// TIA Portal V16 program export: 1 tag tables, 0 data types, 3 data blocks, 1 code blocks (in call order from the OBs), 0 instance data blocks

VAR_GLOBAL   // PLC tag table "Default tag table"
   Web_Integer AT %MW10 : Int;
END_VAR

DATA_BLOCK "Data_block_1"   // DB1
{ S7_Optimized_Access := 'TRUE' }
VERSION : 0.1
// stored: AutoNumber true, DBAccessibleFromOPCUA true, IsOnlyStoredInLoadMemory false, IsRetainMemResEnabled false, IsWriteProtectedInAS false, MemoryReserve 100
   VAR
      in1 : Bool;
      in2 : Bool;
      in3 : Bool;
      out1 : Bool;
      out2 : Bool;
      out3 : Bool;
   END_VAR
BEGIN
END_DATA_BLOCK

DATA_BLOCK "Parameter_Control"   // DB2
{ S7_Optimized_Access := 'TRUE' }
// stored: MemoryReserve 100
   VAR
      Sugar : Real;
      Salt : Int;
      Water : Int;
      Coffee_Powder : Int;
   END_VAR
BEGIN
END_DATA_BLOCK

DATA_BLOCK "Test"   // DB1
{ S7_Optimized_Access := 'TRUE' }
// stored: MemoryReserve 100
   VAR
      testing_bool_output : Bool;
      testing_bool_input : Bool;
      Tag_A : Int := 1;
      Tag_B : Int := 2;
      Tag_C : Int := 3;
      Tag_D : Int := 4;
      Tag_E : Int := 5;
      Testing : Array[0..4] of Int;
   END_VAR
BEGIN
END_DATA_BLOCK

ORGANIZATION_BLOCK "Main"   // OB1, LAD, ProgramCycle
TITLE = "Main Program Sweep (Cycle)"
{ S7_Optimized_Access := 'TRUE' }
VERSION : 0.1
// stored: AutoNumber true, IsIECCheckEnabled false, SetENOAutomatically false
   VAR_INPUT
      Initial_Call : Bool;   // Initial call of this OB
      Remanence : Bool;   // =True, if remanent data are available
   END_VAR
BEGIN

REGION Network 1
   // test demo - v1
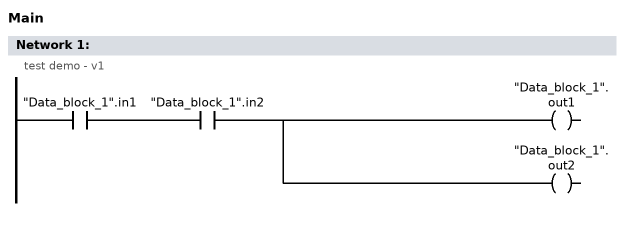
   RUNG wire#powerrail
      Contact( "Data_block_1".in1 )
      Contact( "Data_block_1".in2 )
      wire#w1
      Coil( "Data_block_1".out1 )
   END_RUNG
   RUNG wire#w1
      Coil( "Data_block_1".out2 )
   END_RUNG
   // the same network as SCL:
   "Data_block_1".out1 := "Data_block_1".in1 AND "Data_block_1".in2;
   "Data_block_1".out2 := "Data_block_1".out1;
END_REGION
END_ORGANIZATION_BLOCK
